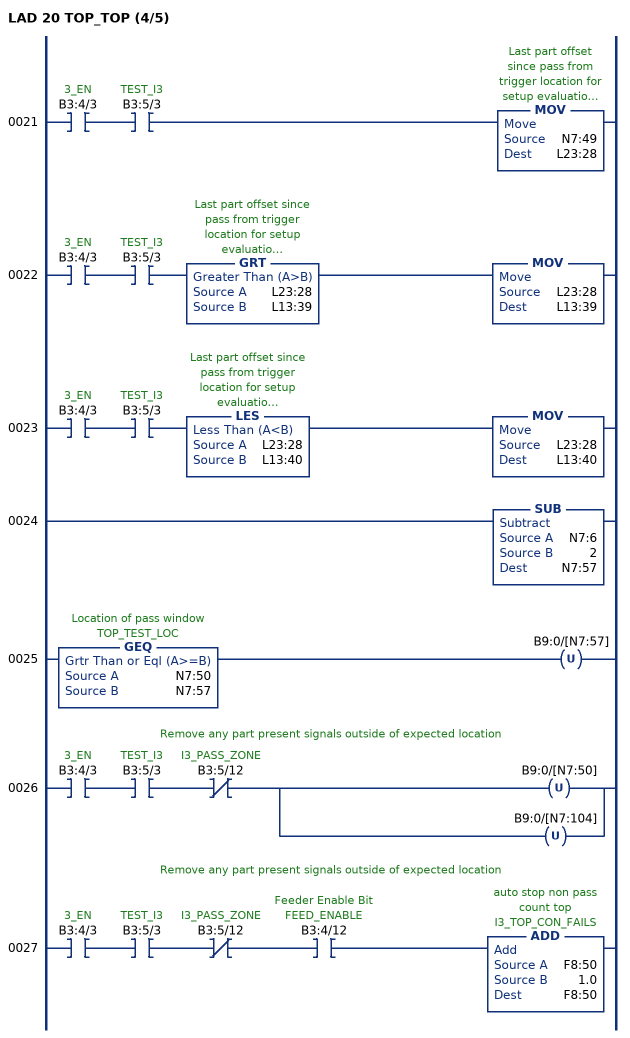
% Rung: 21 %
SOR XIC B3:4/3 XIC B3:5/3 MOV N7:49 L23:28 EOR
%   B3:4/3  3_EN %
%   B3:5/3  TEST_I3 %
%   N7:49  TOP_SINCE_PASS  "distance since top camera pass" %
%   L23:28  LAST_TOP_OFFSET  "Last part offset since pass from trigger location for setup evaluation" %
% Rung: 22 %
SOR XIC B3:4/3 XIC B3:5/3 GRT L23:28 L13:39 MOV L23:28 L13:39 EOR
%   B3:4/3  3_EN %
%   B3:5/3  TEST_I3 %
%   L23:28  LAST_TOP_OFFSET  "Last part offset since pass from trigger location for setup evaluation" %
% Rung: 23 %
SOR XIC B3:4/3 XIC B3:5/3 LES L23:28 L13:40 MOV L23:28 L13:40 EOR
%   B3:4/3  3_EN %
%   B3:5/3  TEST_I3 %
%   L23:28  LAST_TOP_OFFSET  "Last part offset since pass from trigger location for setup evaluation" %
% Rung: 24 %
SOR SUB N7:6 2 N7:57 EOR
%   N7:6  BLOW_LOC_INTEGER  "Blow-off Position" %
% Rung: 25 %
SOR GEQ N7:50 N7:57 OTU B9:0/[N7:57] EOR
%   N7:50  TOP_TEST_LOC  "Location of pass window" %
% Rung: 26 %
% Remove any part present signals outside of expected location %
SOR XIC B3:4/3 XIC B3:5/3 XIO B3:5/12 BST OTU B9:0/[N7:50] NXB OTU B9:0/[N7:104] BND EOR
%   B3:4/3  3_EN %
%   B3:5/3  TEST_I3 %
%   B3:5/12  I3_PASS_ZONE %
%   N7:50  TOP_TEST_LOC  "Location of pass window" %
%   N7:104  2ED_TOP %
% Rung: 27 %
% Remove any part present signals outside of expected location %
SOR XIC B3:4/3 XIC B3:5/3 XIO B3:5/12 XIC B3:4/12 ADD F8:50 1.0 F8:50 EOR
%   B3:4/3  3_EN %
%   B3:5/3  TEST_I3 %
%   B3:5/12  I3_PASS_ZONE %
%   B3:4/12  FEED_ENABLE  "Feeder Enable Bit" %
%   F8:50  I3_TOP_CON_FAILS  "auto stop non pass count top" %

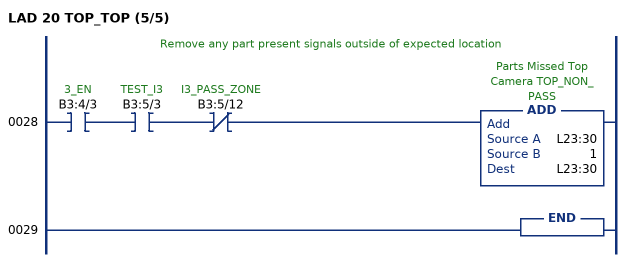
% Rung: 28 %
% Remove any part present signals outside of expected location %
SOR XIC B3:4/3 XIC B3:5/3 XIO B3:5/12 ADD L23:30 1 L23:30 EOR
%   B3:4/3  3_EN %
%   B3:5/3  TEST_I3 %
%   B3:5/12  I3_PASS_ZONE %
%   L23:30  TOP_NON_PASS  "Parts Missed Top Camera" %
% Rung: 29 %
SOR END EOR

LADDER 24 "TOP_BLOW"
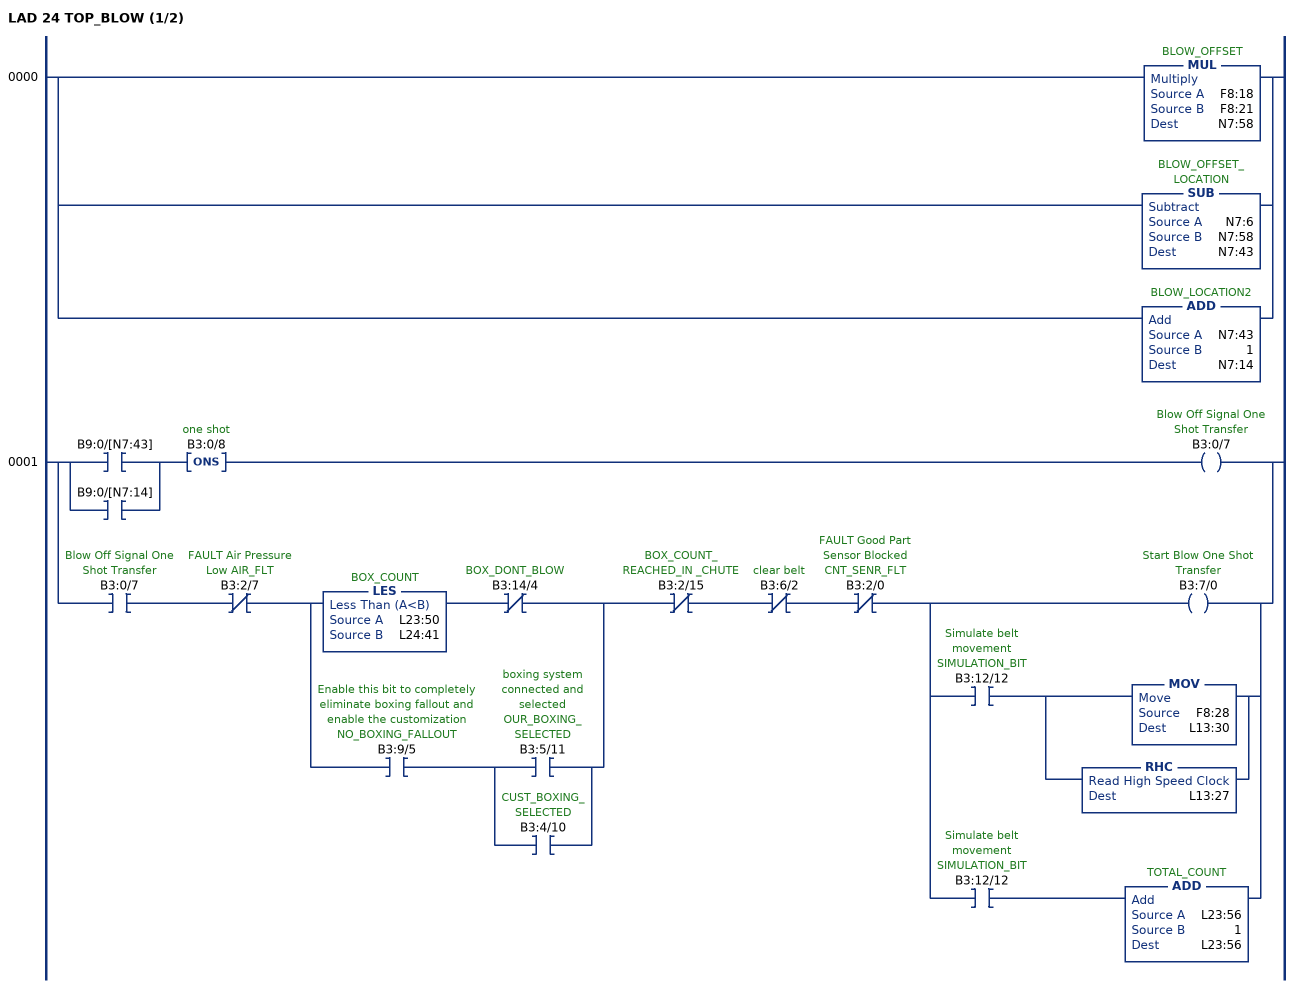
% Rung: 0 %
SOR BST MUL F8:18 F8:21 N7:58 NXB SUB N7:6 N7:58 N7:43 NXB ADD N7:43 1 N7:14 BND EOR
%   F8:18  TOP_SPEED  "top belt speed average in pulses per second 290 Max; Verify" %
%   F8:21  BLOW_COMP_TIME %
%   N7:58  BLOW_OFFSET %
%   N7:6  BLOW_LOC_INTEGER  "Blow-off Position" %
%   N7:43  BLOW_OFFSET_LOCATION %
%   N7:14  BLOW_LOCATION2 %
% Rung: 1 %
SOR BST BST XIC B9:0/[N7:43] NXB XIC B9:0/[N7:14] BND ONS B3:0/8 OTE B3:0/7 NXB XIC B3:0/7 XIO B3:2/7 BST LES L23:50 L24:41 XIO B3:14/4 NXB XIC B3:9/5 BST XIC B3:5/11 NXB XIC B3:4/10 BND BND XIO B3:2/15 XIO B3:6/2 XIO B3:2/0 BST OTE B3:7/0 NXB XIC B3:12/12 BST MOV F8:28 L13:30 NXB RHC L13:27 BND NXB XIC B3:12/12 ADD L23:56 1 L23:56 BND BND EOR
%   N7:43  BLOW_OFFSET_LOCATION %
%   N7:14  BLOW_LOCATION2 %
%   B3:0/8  "one shot" %
%   B3:0/7  "Blow Off Signal One Shot Transfer" %
%   B3:2/7  AIR_FLT  "FAULT Air Pressure Low" %
%   L23:50  BOX_COUNT %
%   L24:41  BOX_COUNT_LIMIT %
%   B3:14/4  BOX_DONT_BLOW %
%   B3:9/5  NO_BOXING_FALLOUT  "Enable this bit to completely eliminate boxing fallout and enable the customization" %
%   B3:5/11  OUR_BOXING_SELECTED  "boxing system connected and selected" %
%   B3:4/10  CUST_BOXING_SELECTED %
%   B3:2/15  "BOX_COUNT_REACHED_IN _CHUTE" %
%   B3:6/2  "clear belt" %
%   B3:2/0  CNT_SENR_FLT  "FAULT Good Part Sensor Blocked" %
%   B3:7/0  "Start Blow One Shot Transfer" %
%   B3:12/12  SIMULATION_BIT  "Simulate belt movement" %
%   F8:28  "momentary rate in ppm" %
%   L23:56  TOTAL_COUNT %

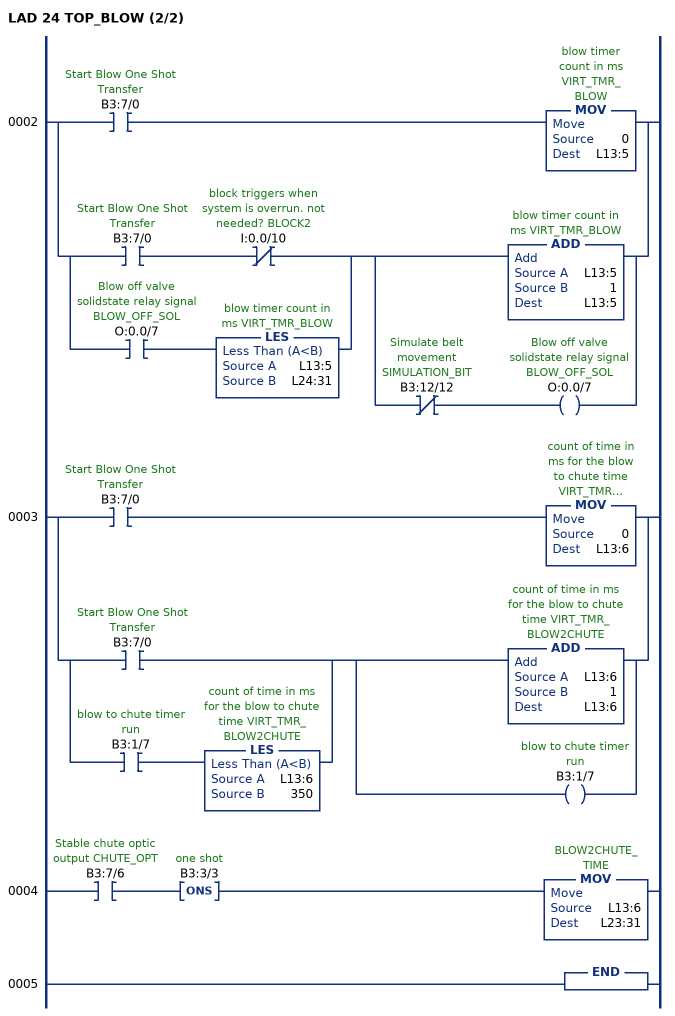
% Rung: 2 %
SOR BST XIC B3:7/0 MOV 0 L13:5 NXB BST XIC B3:7/0 XIO I:0.0/10 NXB XIC O:0.0/7 LES L13:5 L24:31 BND BST ADD L13:5 1 L13:5 NXB XIO B3:12/12 OTE O:0.0/7 BND BND EOR
%   B3:7/0  "Start Blow One Shot Transfer" %
%   L13:5  VIRT_TMR_BLOW  "blow timer count in ms" %
%   I:0.0/10  BLOCK2  "block triggers when system is overrun. not needed?" %
%   O:0.0/7  BLOW_OFF_SOL  "Blow off valve solidstate relay signal" %
%   L24:31  BLOW_TIME %
%   B3:12/12  SIMULATION_BIT  "Simulate belt movement" %
% Rung: 3 %
SOR BST XIC B3:7/0 MOV 0 L13:6 NXB BST XIC B3:7/0 NXB XIC B3:1/7 LES L13:6 350 BND BST ADD L13:6 1 L13:6 NXB OTE B3:1/7 BND BND EOR
%   B3:7/0  "Start Blow One Shot Transfer" %
%   L13:6  VIRT_TMR_BLOW2CHUTE  "count of time in ms for the blow to chute time" %
%   B3:1/7  "blow to chute timer run" %
% Rung: 4 %
SOR XIC B3:7/6 ONS B3:3/3 MOV L13:6 L23:31 EOR
%   B3:7/6  CHUTE_OPT  "Stable chute optic output" %
%   B3:3/3  "one shot" %
%   L13:6  VIRT_TMR_BLOW2CHUTE  "count of time in ms for the blow to chute time" %
%   L23:31  BLOW2CHUTE_TIME %
% Rung: 5 %
SOR END EOR

LADDER 28 "FAULTS"
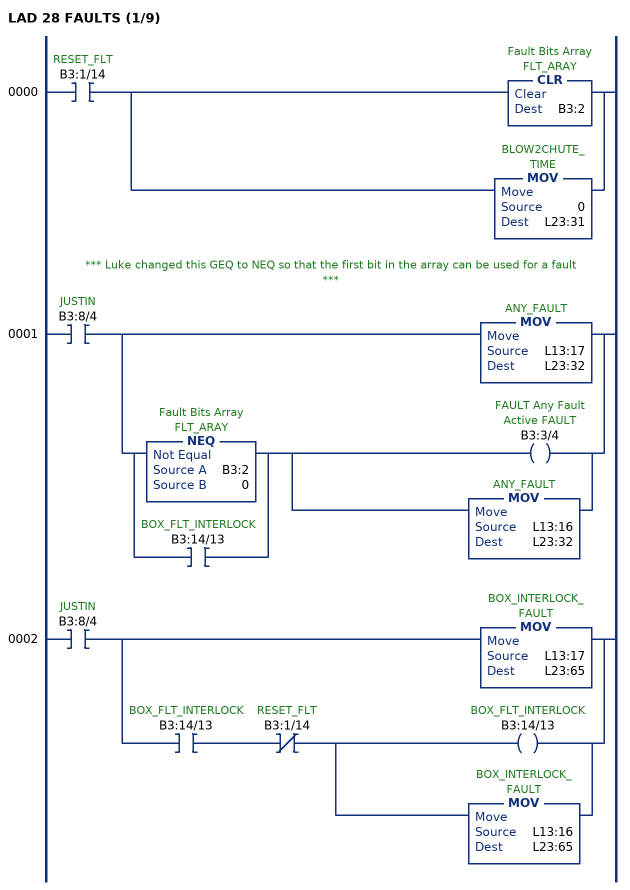
% Rung: 0 %
SOR XIC B3:1/14 BST CLR B3:2 NXB MOV 0 L23:31 BND EOR
%   B3:1/14  RESET_FLT %
%   B3:2  FLT_ARAY  "Fault Bits Array" %
%   L23:31  BLOW2CHUTE_TIME %
% Rung: 1 %
% *** Luke changed this GEQ to NEQ so that the first bit in the array can be used for a fault *** %
SOR XIC B3:8/4 BST MOV L13:17 L23:32 NXB BST NEQ B3:2 0 NXB XIC B3:14/13 BND BST OTE B3:3/4 NXB MOV L13:16 L23:32 BND BND EOR
%   B3:8/4  JUSTIN %
%   L13:17  FALSE %
%   L23:32  ANY_FAULT %
%   B3:2  FLT_ARAY  "Fault Bits Array" %
%   B3:14/13  BOX_FLT_INTERLOCK %
%   B3:3/4  FAULT  "FAULT Any Fault Active" %
%   L13:16  TRUE  "ONE TIME ENABLE FOR THE TIMES WHEN WE FORGET TO RE-ENABLE AFTER SHIPMENT" %
% Rung: 2 %
SOR XIC B3:8/4 BST MOV L13:17 L23:65 NXB XIC B3:14/13 XIO B3:1/14 BST OTE B3:14/13 NXB MOV L13:16 L23:65 BND BND EOR
%   B3:8/4  JUSTIN %
%   L13:17  FALSE %
%   L23:65  BOX_INTERLOCK_FAULT %
%   B3:14/13  BOX_FLT_INTERLOCK %
%   B3:1/14  RESET_FLT %
%   L13:16  TRUE  "ONE TIME ENABLE FOR THE TIMES WHEN WE FORGET TO RE-ENABLE AFTER SHIPMENT" %

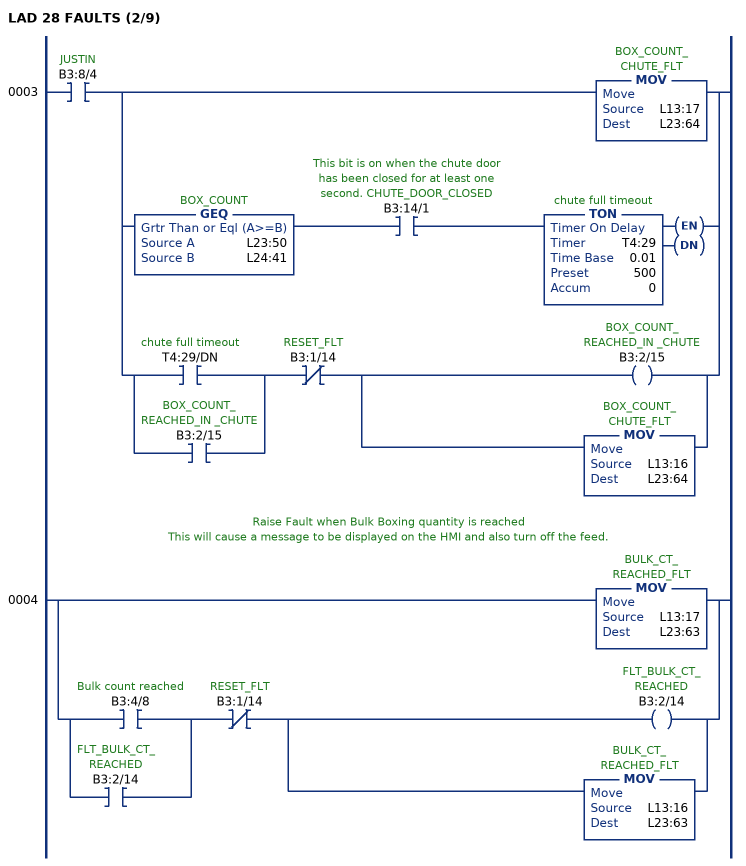
% Rung: 3 %
SOR XIC B3:8/4 BST MOV L13:17 L23:64 NXB GEQ L23:50 L24:41 XIC B3:14/1 TON T4:29 0.01 500 0 NXB BST XIC T4:29/DN NXB XIC B3:2/15 BND XIO B3:1/14 BST OTE B3:2/15 NXB MOV L13:16 L23:64 BND BND EOR
%   B3:8/4  JUSTIN %
%   L13:17  FALSE %
%   L23:64  BOX_COUNT_CHUTE_FLT %
%   L23:50  BOX_COUNT %
%   L24:41  BOX_COUNT_LIMIT %
%   B3:14/1  CHUTE_DOOR_CLOSED  "This bit is on when the chute door has been closed for at least one second." %
%   T4:29  "chute full timeout" %
%   B3:2/15  "BOX_COUNT_REACHED_IN _CHUTE" %
%   B3:1/14  RESET_FLT %
%   L13:16  TRUE  "ONE TIME ENABLE FOR THE TIMES WHEN WE FORGET TO RE-ENABLE AFTER SHIPMENT" %
% Rung: 4 %
% Raise Fault when Bulk Boxing quantity is reached
% 
% This will cause a message to be displayed on the HMI and also turn off the feed. %
SOR BST MOV L13:17 L23:63 NXB BST XIC B3:4/8 NXB XIC B3:2/14 BND XIO B3:1/14 BST OTE B3:2/14 NXB MOV L13:16 L23:63 BND BND EOR
%   L13:17  FALSE %
%   L23:63  BULK_CT_REACHED_FLT %
%   B3:4/8  "Bulk count reached" %
%   B3:2/14  FLT_BULK_CT_REACHED %
%   B3:1/14  RESET_FLT %
%   L13:16  TRUE  "ONE TIME ENABLE FOR THE TIMES WHEN WE FORGET TO RE-ENABLE AFTER SHIPMENT" %

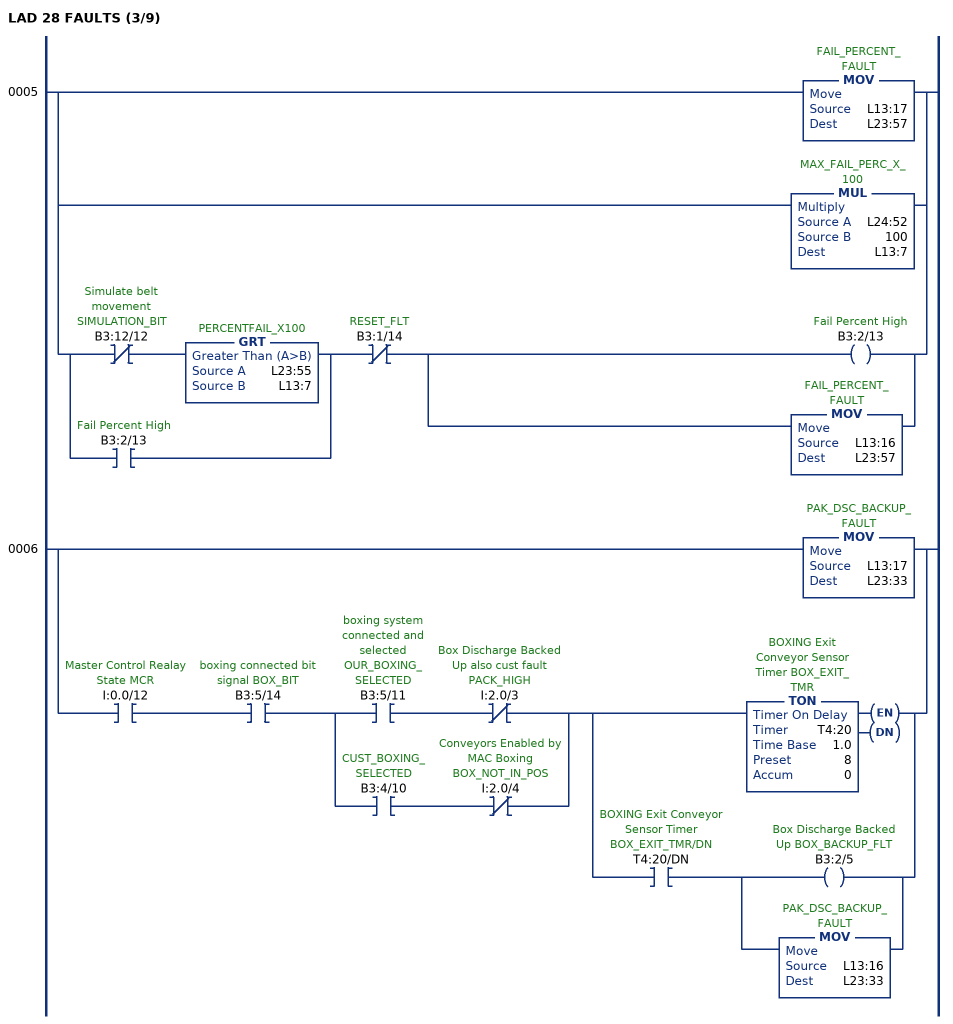
% Rung: 5 %
SOR BST MOV L13:17 L23:57 NXB MUL L24:52 100 L13:7 NXB BST XIO B3:12/12 GRT L23:55 L13:7 NXB XIC B3:2/13 BND XIO B3:1/14 BST OTE B3:2/13 NXB MOV L13:16 L23:57 BND BND EOR
%   L13:17  FALSE %
%   L23:57  FAIL_PERCENT_FAULT %
%   L24:52  MAX_FAIL_PERCENT %
%   L13:7  MAX_FAIL_PERC_X_100 %
%   B3:12/12  SIMULATION_BIT  "Simulate belt movement" %
%   L23:55  PERCENTFAIL_X100 %
%   B3:2/13  "Fail Percent High" %
%   B3:1/14  RESET_FLT %
%   L13:16  TRUE  "ONE TIME ENABLE FOR THE TIMES WHEN WE FORGET TO RE-ENABLE AFTER SHIPMENT" %
% Rung: 6 %
SOR BST MOV L13:17 L23:33 NXB XIC I:0.0/12 XIC B3:5/14 BST XIC B3:5/11 XIO I:2.0/3 NXB XIC B3:4/10 XIO I:2.0/4 BND BST TON T4:20 1.0 8 0 NXB XIC T4:20/DN BST OTE B3:2/5 NXB MOV L13:16 L23:33 BND BND BND EOR
%   L13:17  FALSE %
%   L23:33  PAK_DSC_BACKUP_FAULT %
%   I:0.0/12  MCR  "Master Control Realay State" %
%   B3:5/14  BOX_BIT  "boxing connected bit signal" %
%   B3:5/11  OUR_BOXING_SELECTED  "boxing system connected and selected" %
%   I:2.0/3  PACK_HIGH  "Box Discharge Backed Up also cust fault" %
%   B3:4/10  CUST_BOXING_SELECTED %
%   I:2.0/4  BOX_NOT_IN_POS  "Conveyors Enabled by MAC Boxing" %
%   T4:20  BOX_EXIT_TMR  "BOXING Exit Conveyor Sensor Timer" %
%   B3:2/5  BOX_BACKUP_FLT  "Box Discharge Backed Up" %
%   L13:16  TRUE  "ONE TIME ENABLE FOR THE TIMES WHEN WE FORGET TO RE-ENABLE AFTER SHIPMENT" %

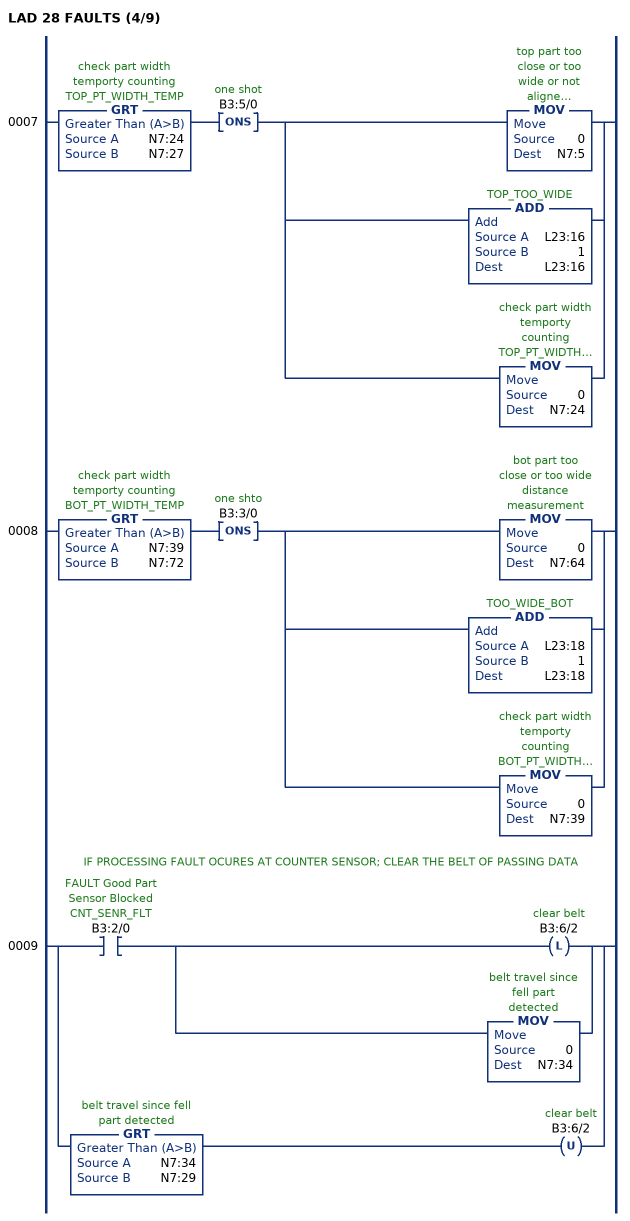
% Rung: 7 %
SOR GRT N7:24 N7:27 ONS B3:5/0 BST MOV 0 N7:5 NXB ADD L23:16 1 L23:16 NXB MOV 0 N7:24 BND EOR
%   N7:24  TOP_PT_WIDTH_TEMP  "check part width temporty counting" %
%   N7:27  "max part width top optic" %
%   B3:5/0  "one shot" %
%   N7:5  "top part too close or too wide or not aligned distance measurement" %
%   L23:16  TOP_TOO_WIDE %
% Rung: 8 %
SOR GRT N7:39 N7:72 ONS B3:3/0 BST MOV 0 N7:64 NXB ADD L23:18 1 L23:18 NXB MOV 0 N7:39 BND EOR
%   N7:39  BOT_PT_WIDTH_TEMP  "check part width temporty counting" %
%   N7:72  "max part width bottom optic" %
%   B3:3/0  "one shto" %
%   N7:64  "bot part too close or too wide distance measurement" %
%   L23:18  TOO_WIDE_BOT %
% Rung: 9 %
% IF PROCESSING FAULT OCURES AT COUNTER SENSOR; CLEAR THE BELT OF PASSING DATA %
SOR BST XIC B3:2/0 BST OTL B3:6/2 NXB MOV 0 N7:34 BND NXB GRT N7:34 N7:29 OTU B3:6/2 BND EOR
%   B3:2/0  CNT_SENR_FLT  "FAULT Good Part Sensor Blocked" %
%   B3:6/2  "clear belt" %
%   N7:34  "belt travel since fell part detected" %
%   N7:29  "belt travel to wipe parts off of belt when fell part detected" %

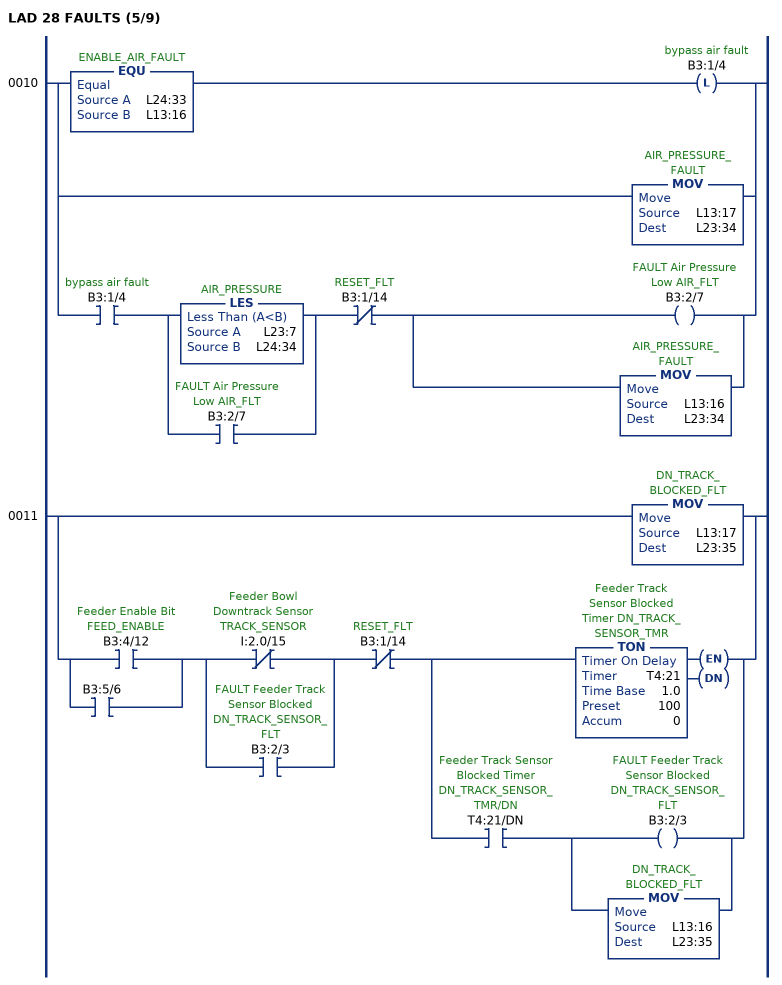
% Rung: 10 %
SOR BST EQU L24:33 L13:16 OTL B3:1/4 NXB MOV L13:17 L23:34 NXB XIC B3:1/4 BST LES L23:7 L24:34 NXB XIC B3:2/7 BND XIO B3:1/14 BST OTE B3:2/7 NXB MOV L13:16 L23:34 BND BND EOR
%   L24:33  ENABLE_AIR_FAULT %
%   L13:16  TRUE  "ONE TIME ENABLE FOR THE TIMES WHEN WE FORGET TO RE-ENABLE AFTER SHIPMENT" %
%   B3:1/4  "bypass air fault" %
%   L13:17  FALSE %
%   L23:34  AIR_PRESSURE_FAULT %
%   L23:7  AIR_PRESSURE %
%   L24:34  MIN_AIR_PRESSURE %
%   B3:2/7  AIR_FLT  "FAULT Air Pressure Low" %
%   B3:1/14  RESET_FLT %
% Rung: 11 %
SOR BST MOV L13:17 L23:35 NXB BST XIC B3:4/12 NXB XIC B3:5/6 BND BST XIO I:2.0/15 NXB XIC B3:2/3 BND XIO B3:1/14 BST TON T4:21 1.0 100 0 NXB XIC T4:21/DN BST OTE B3:2/3 NXB MOV L13:16 L23:35 BND BND BND EOR
%   L13:17  FALSE %
%   L23:35  DN_TRACK_BLOCKED_FLT %
%   B3:4/12  FEED_ENABLE  "Feeder Enable Bit" %
%   I:2.0/15  TRACK_SENSOR  "Feeder Bowl Downtrack Sensor" %
%   B3:2/3  DN_TRACK_SENSOR_FLT  "FAULT Feeder Track Sensor Blocked" %
%   B3:1/14  RESET_FLT %
%   T4:21  DN_TRACK_SENSOR_TMR  "Feeder Track Sensor Blocked Timer" %
%   L13:16  TRUE  "ONE TIME ENABLE FOR THE TIMES WHEN WE FORGET TO RE-ENABLE AFTER SHIPMENT" %

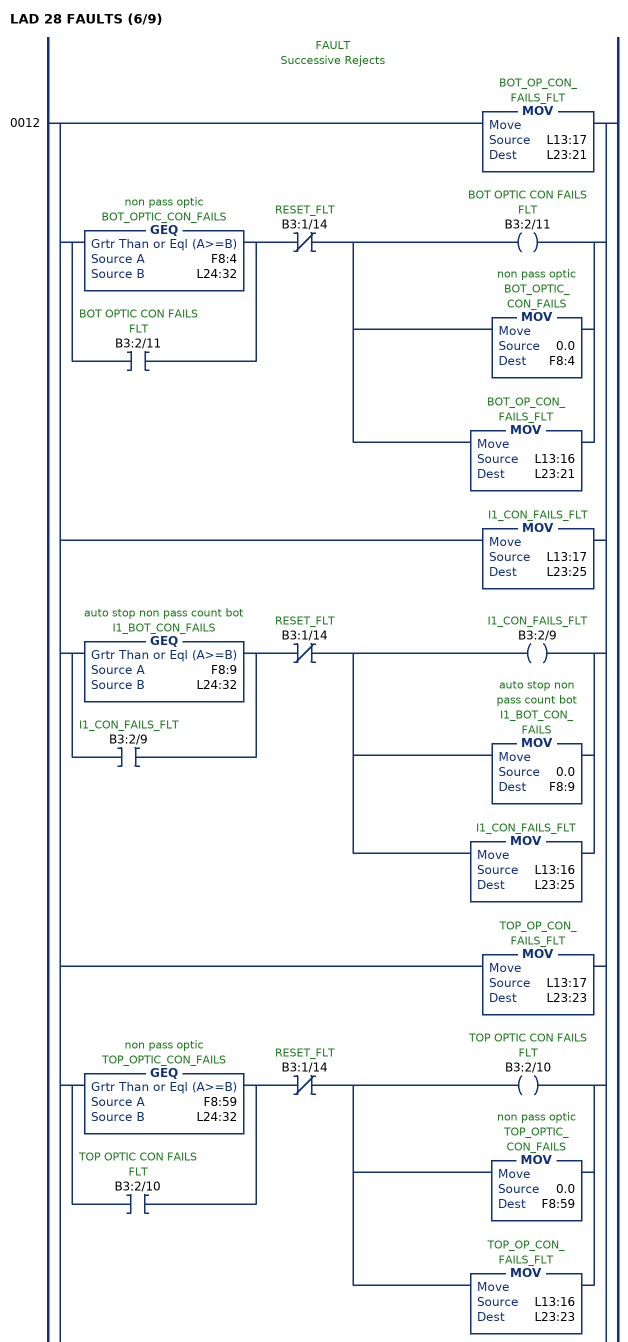

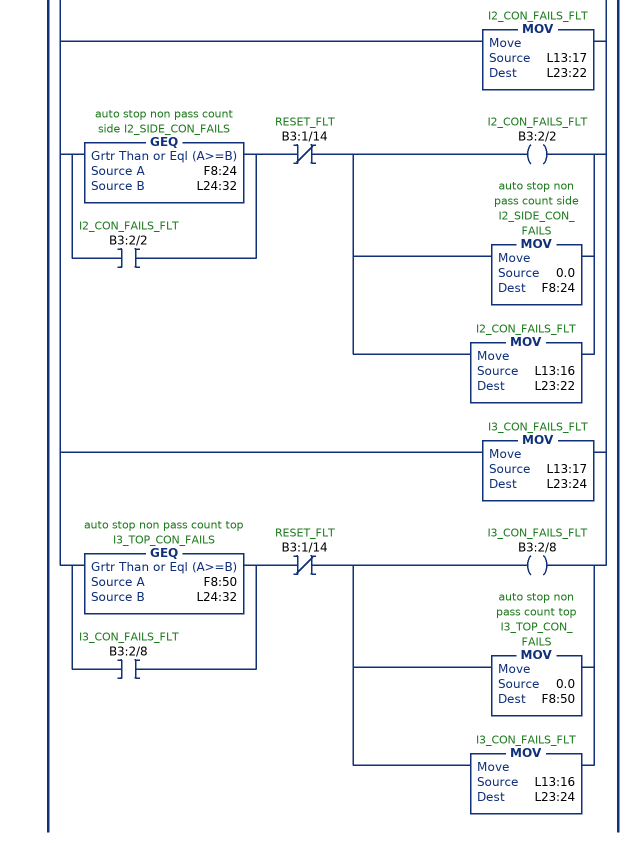
% Rung: 12 %
% FAULT
% Successive Rejects %
SOR BST BST MOV L13:17 L23:21 NXB BST GEQ F8:4 L24:32 NXB XIC B3:2/11 BND XIO B3:1/14 BST OTE B3:2/11 NXB MOV 0.0 F8:4 NXB MOV L13:16 L23:21 BND BND NXB BST MOV L13:17 L23:25 NXB BST GEQ F8:9 L24:32 NXB XIC B3:2/9 BND XIO B3:1/14 BST OTE B3:2/9 NXB MOV 0.0 F8:9 NXB MOV L13:16 L23:25 BND BND NXB BST MOV L13:17 L23:23 NXB BST GEQ F8:59 L24:32 NXB XIC B3:2/10 BND XIO B3:1/14 BST OTE B3:2/10 NXB MOV 0.0 F8:59 NXB MOV L13:16 L23:23 BND BND NXB BST MOV L13:17 L23:22 NXB BST GEQ F8:24 L24:32 NXB XIC B3:2/2 BND XIO B3:1/14 BST OTE B3:2/2 NXB MOV 0.0 F8:24 NXB MOV L13:16 L23:22 BND BND NXB BST MOV L13:17 L23:24 NXB BST GEQ F8:50 L24:32 NXB XIC B3:2/8 BND XIO B3:1/14 BST OTE B3:2/8 NXB MOV 0.0 F8:50 NXB MOV L13:16 L23:24 BND BND BND EOR
%   L13:17  FALSE %
%   L23:21  BOT_OP_CON_FAILS_FLT %
%   F8:4  BOT_OPTIC_CON_FAILS  "non pass optic" %
%   L24:32  MAX_CON_FAILS %
%   B3:2/11  "BOT OPTIC CON FAILS FLT" %
%   B3:1/14  RESET_FLT %
%   L13:16  TRUE  "ONE TIME ENABLE FOR THE TIMES WHEN WE FORGET TO RE-ENABLE AFTER SHIPMENT" %
%   L23:25  I1_CON_FAILS_FLT %
%   F8:9  I1_BOT_CON_FAILS  "auto stop non pass count bot" %
%   B3:2/9  "I1_CON_FAILS_FLT" %
%   L23:23  TOP_OP_CON_FAILS_FLT %
%   F8:59  TOP_OPTIC_CON_FAILS  "non pass optic" %
%   B3:2/10  "TOP OPTIC CON FAILS FLT" %
%   L23:22  I2_CON_FAILS_FLT %
%   F8:24  I2_SIDE_CON_FAILS  "auto stop non pass count side" %
%   B3:2/2  "I2_CON_FAILS_FLT" %
%   L23:24  I3_CON_FAILS_FLT %
%   F8:50  I3_TOP_CON_FAILS  "auto stop non pass count top" %
%   B3:2/8  "I3_CON_FAILS_FLT" %

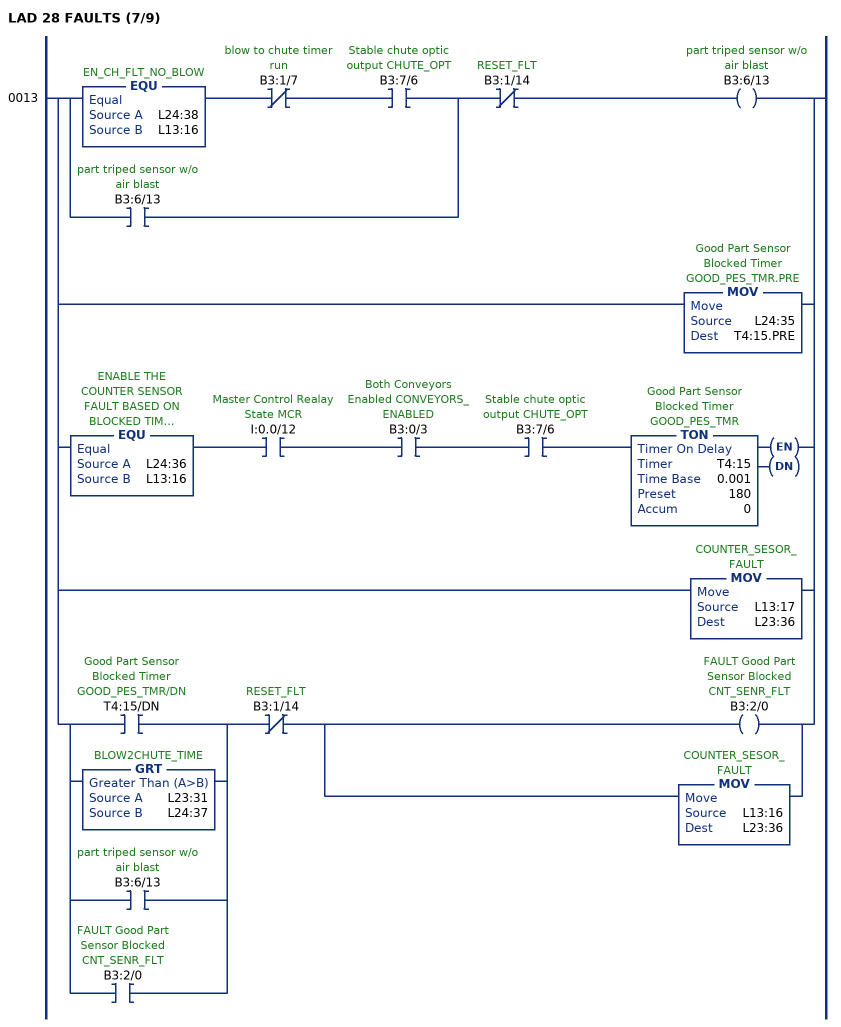
% Rung: 13 %
SOR BST BST EQU L24:38 L13:16 XIO B3:1/7 XIC B3:7/6 NXB XIC B3:6/13 BND XIO B3:1/14 OTE B3:6/13 NXB MOV L24:35 T4:15.PRE NXB EQU L24:36 L13:16 XIC I:0.0/12 XIC B3:0/3 XIC B3:7/6 TON T4:15 0.001 180 0 NXB MOV L13:17 L23:36 NXB BST XIC T4:15/DN NXB GRT L23:31 L24:37 NXB XIC B3:6/13 NXB XIC B3:2/0 BND XIO B3:1/14 BST OTE B3:2/0 NXB MOV L13:16 L23:36 BND BND EOR
%   L24:38  EN_CH_FLT_NO_BLOW %
%   L13:16  TRUE  "ONE TIME ENABLE FOR THE TIMES WHEN WE FORGET TO RE-ENABLE AFTER SHIPMENT" %
%   B3:1/7  "blow to chute timer run" %
%   B3:7/6  CHUTE_OPT  "Stable chute optic output" %
%   B3:6/13  "part triped sensor w/o air blast" %
%   B3:1/14  RESET_FLT %
%   L24:35  GD_PT_SEN_BLKED_TM %
%   T4:15  GOOD_PES_TMR  "Good Part Sensor Blocked Timer" %
%   L24:36  EN_CT_BL_TM_FAULT  "ENABLE THE COUNTER SENSOR FAULT BASED ON BLOCKED TIME" %
%   I:0.0/12  MCR  "Master Control Realay State" %
%   B3:0/3  CONVEYORS_ENABLED  "Both Conveyors Enabled" %
%   L13:17  FALSE %
%   L23:36  COUNTER_SESOR_FAULT %
%   L23:31  BLOW2CHUTE_TIME %
%   L24:37  MAX_BLOW2CHUTE_MS %
%   B3:2/0  CNT_SENR_FLT  "FAULT Good Part Sensor Blocked" %

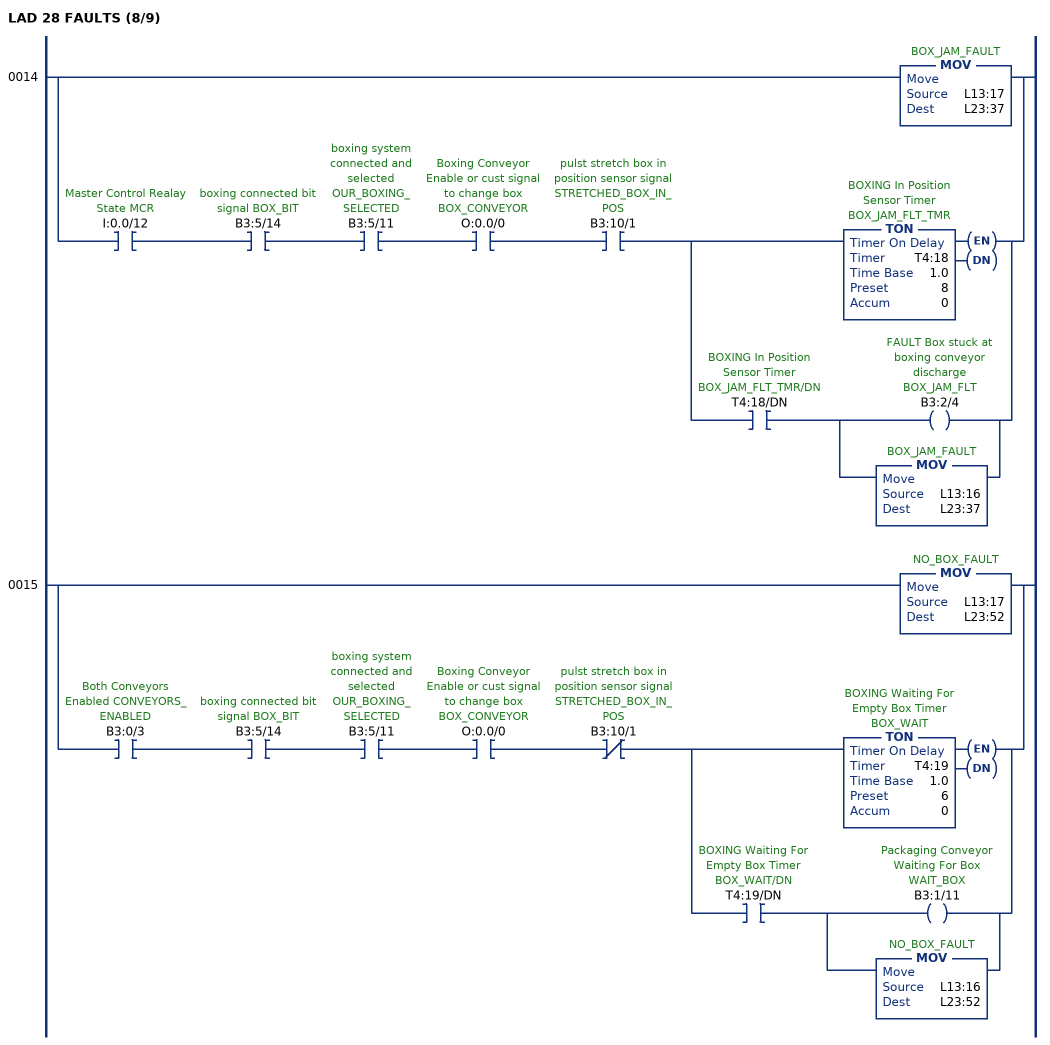
% Rung: 14 %
SOR BST MOV L13:17 L23:37 NXB XIC I:0.0/12 XIC B3:5/14 XIC B3:5/11 XIC O:0.0/0 XIC B3:10/1 BST TON T4:18 1.0 8 0 NXB XIC T4:18/DN BST OTE B3:2/4 NXB MOV L13:16 L23:37 BND BND BND EOR
%   L13:17  FALSE %
%   L23:37  BOX_JAM_FAULT %
%   I:0.0/12  MCR  "Master Control Realay State" %
%   B3:5/14  BOX_BIT  "boxing connected bit signal" %
%   B3:5/11  OUR_BOXING_SELECTED  "boxing system connected and selected" %
%   O:0.0/0  BOX_CONVEYOR  "Boxing Conveyor Enable or cust signal to change box" %
%   B3:10/1  STRETCHED_BOX_IN_POS  "pulst stretch box in position sensor signal" %
%   T4:18  BOX_JAM_FLT_TMR  "BOXING In Position Sensor Timer" %
%   B3:2/4  BOX_JAM_FLT  "FAULT Box stuck at boxing conveyor discharge" %
%   L13:16  TRUE  "ONE TIME ENABLE FOR THE TIMES WHEN WE FORGET TO RE-ENABLE AFTER SHIPMENT" %
% Rung: 15 %
SOR BST MOV L13:17 L23:52 NXB XIC B3:0/3 XIC B3:5/14 XIC B3:5/11 XIC O:0.0/0 XIO B3:10/1 BST TON T4:19 1.0 6 0 NXB XIC T4:19/DN BST OTE B3:1/11 NXB MOV L13:16 L23:52 BND BND BND EOR
%   L13:17  FALSE %
%   L23:52  NO_BOX_FAULT %
%   B3:0/3  CONVEYORS_ENABLED  "Both Conveyors Enabled" %
%   B3:5/14  BOX_BIT  "boxing connected bit signal" %
%   B3:5/11  OUR_BOXING_SELECTED  "boxing system connected and selected" %
%   O:0.0/0  BOX_CONVEYOR  "Boxing Conveyor Enable or cust signal to change box" %
%   B3:10/1  STRETCHED_BOX_IN_POS  "pulst stretch box in position sensor signal" %
%   T4:19  BOX_WAIT  "BOXING Waiting For Empty Box Timer" %
%   B3:1/11  WAIT_BOX  "Packaging Conveyor Waiting For Box" %
%   L13:16  TRUE  "ONE TIME ENABLE FOR THE TIMES WHEN WE FORGET TO RE-ENABLE AFTER SHIPMENT" %

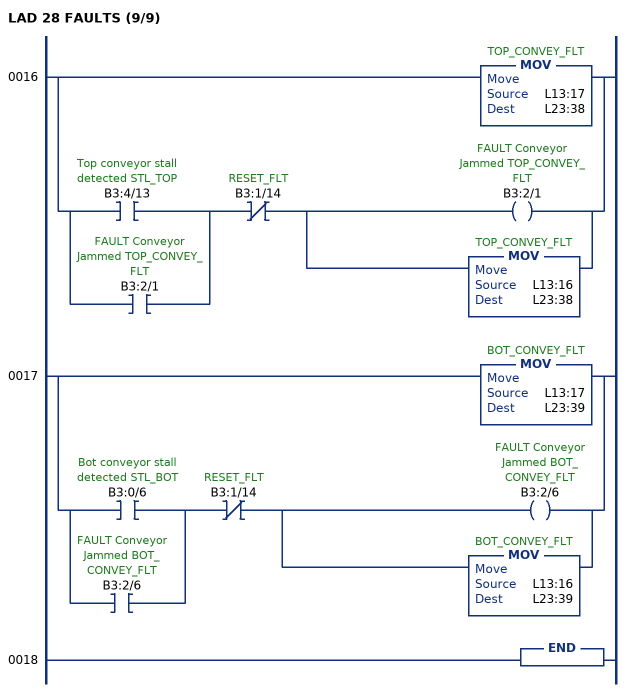
% Rung: 16 %
SOR BST MOV L13:17 L23:38 NXB BST XIC B3:4/13 NXB XIC B3:2/1 BND XIO B3:1/14 BST OTE B3:2/1 NXB MOV L13:16 L23:38 BND BND EOR
%   L13:17  FALSE %
%   L23:38  TOP_CONVEY_FLT %
%   B3:4/13  STL_TOP  "Top conveyor stall detected" %
%   B3:2/1  "FAULT Conveyor Jammed TOP_CONVEY_FLT" %
%   B3:1/14  RESET_FLT %
%   L13:16  TRUE  "ONE TIME ENABLE FOR THE TIMES WHEN WE FORGET TO RE-ENABLE AFTER SHIPMENT" %
% Rung: 17 %
SOR BST MOV L13:17 L23:39 NXB BST XIC B3:0/6 NXB XIC B3:2/6 BND XIO B3:1/14 BST OTE B3:2/6 NXB MOV L13:16 L23:39 BND BND EOR
%   L13:17  FALSE %
%   L23:39  BOT_CONVEY_FLT %
%   B3:0/6  STL_BOT  "Bot conveyor stall detected" %
%   B3:2/6  "FAULT Conveyor Jammed BOT_CONVEY_FLT" %
%   B3:1/14  RESET_FLT %
%   L13:16  TRUE  "ONE TIME ENABLE FOR THE TIMES WHEN WE FORGET TO RE-ENABLE AFTER SHIPMENT" %
% Rung: 18 %
SOR END EOR

LADDER 29 "SPEED"
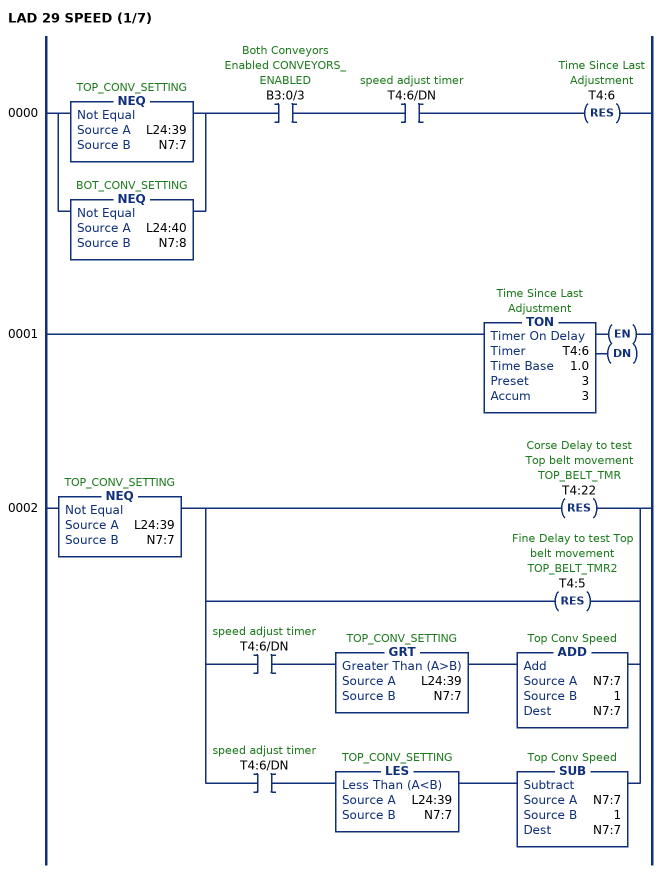
% Rung: 0 %
SOR BST NEQ L24:39 N7:7 NXB NEQ L24:40 N7:8 BND XIC B3:0/3 XIC T4:6/DN RES T4:6 EOR
%   L24:39  TOP_CONV_SETTING %
%   N7:7  "Top Conv Speed" %
%   L24:40  BOT_CONV_SETTING %
%   N7:8  "Bottom Conveyor Speed" %
%   B3:0/3  CONVEYORS_ENABLED  "Both Conveyors Enabled" %
%   T4:6/DN  "speed adjust timer" %
%   T4:6  "Time Since Last Adjustment" %
% Rung: 1 %
SOR TON T4:6 1.0 3 3 EOR
%   T4:6  "Time Since Last Adjustment" %
% Rung: 2 %
SOR NEQ L24:39 N7:7 BST RES T4:22 NXB RES T4:5 NXB XIC T4:6/DN GRT L24:39 N7:7 ADD N7:7 1 N7:7 NXB XIC T4:6/DN LES L24:39 N7:7 SUB N7:7 1 N7:7 BND EOR
%   L24:39  TOP_CONV_SETTING %
%   N7:7  "Top Conv Speed" %
%   T4:22  TOP_BELT_TMR  "Corse Delay to test Top belt movement" %
%   T4:5  TOP_BELT_TMR2  "Fine Delay to test Top belt movement" %
%   T4:6/DN  "speed adjust timer" %

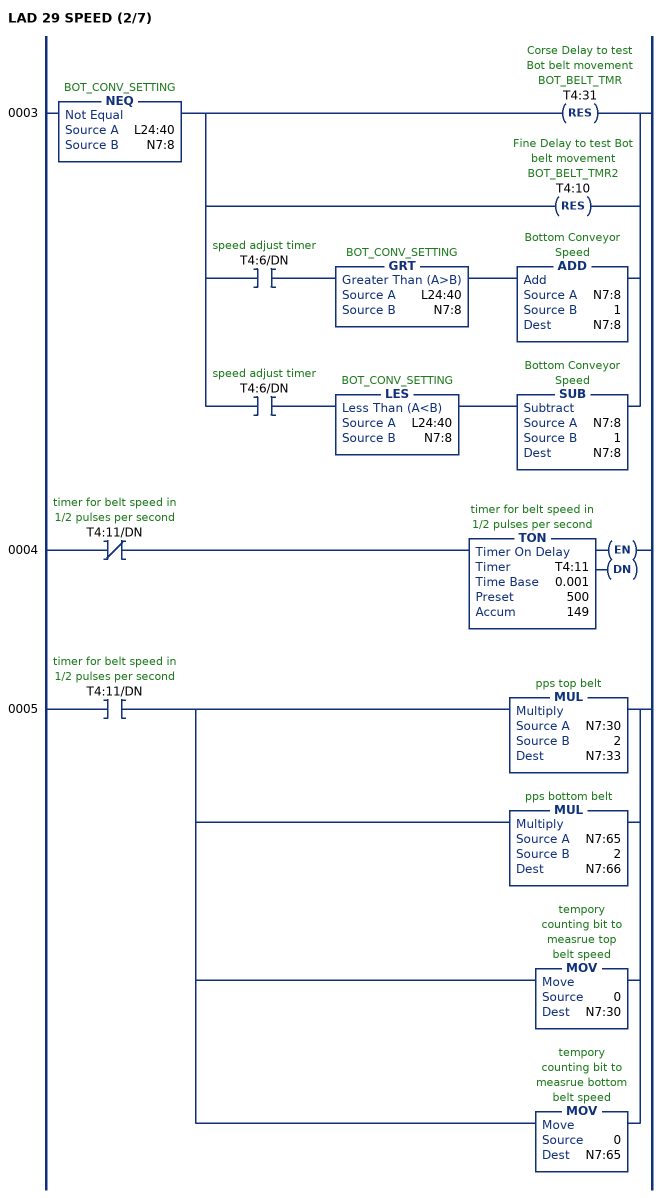
% Rung: 3 %
SOR NEQ L24:40 N7:8 BST RES T4:31 NXB RES T4:10 NXB XIC T4:6/DN GRT L24:40 N7:8 ADD N7:8 1 N7:8 NXB XIC T4:6/DN LES L24:40 N7:8 SUB N7:8 1 N7:8 BND EOR
%   L24:40  BOT_CONV_SETTING %
%   N7:8  "Bottom Conveyor Speed" %
%   T4:31  BOT_BELT_TMR  "Corse Delay to test Bot belt movement" %
%   T4:10  BOT_BELT_TMR2  "Fine Delay to test Bot belt movement" %
%   T4:6/DN  "speed adjust timer" %
% Rung: 4 %
SOR XIO T4:11/DN TON T4:11 0.001 500 149 EOR
%   T4:11  "timer for belt speed in 1/2 pulses per second" %
% Rung: 5 %
SOR XIC T4:11/DN BST MUL N7:30 2 N7:33 NXB MUL N7:65 2 N7:66 NXB MOV 0 N7:30 NXB MOV 0 N7:65 BND EOR
%   T4:11  "timer for belt speed in 1/2 pulses per second" %
%   N7:30  "tempory counting bit to measrue top belt speed" %
%   N7:33  "pps top belt" %
%   N7:65  "tempory counting bit to measrue bottom belt speed" %
%   N7:66  "pps bottom belt" %

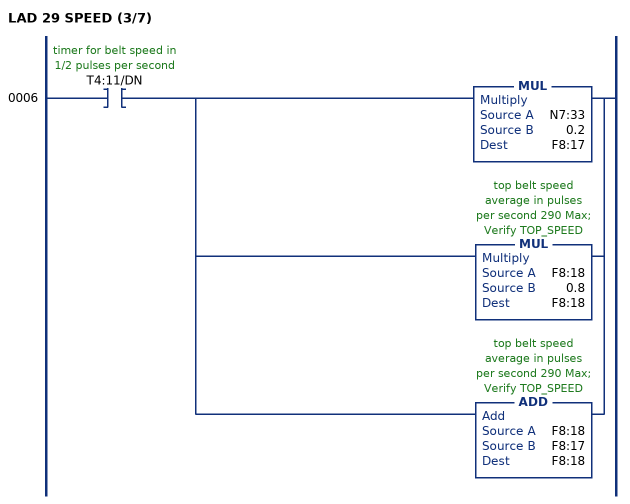
% Rung: 6 %
SOR XIC T4:11/DN BST MUL N7:33 0.2 F8:17 NXB MUL F8:18 0.8 F8:18 NXB ADD F8:18 F8:17 F8:18 BND EOR
%   T4:11  "timer for belt speed in 1/2 pulses per second" %
%   N7:33  "pps top belt" %
%   F8:18  TOP_SPEED  "top belt speed average in pulses per second 290 Max; Verify" %

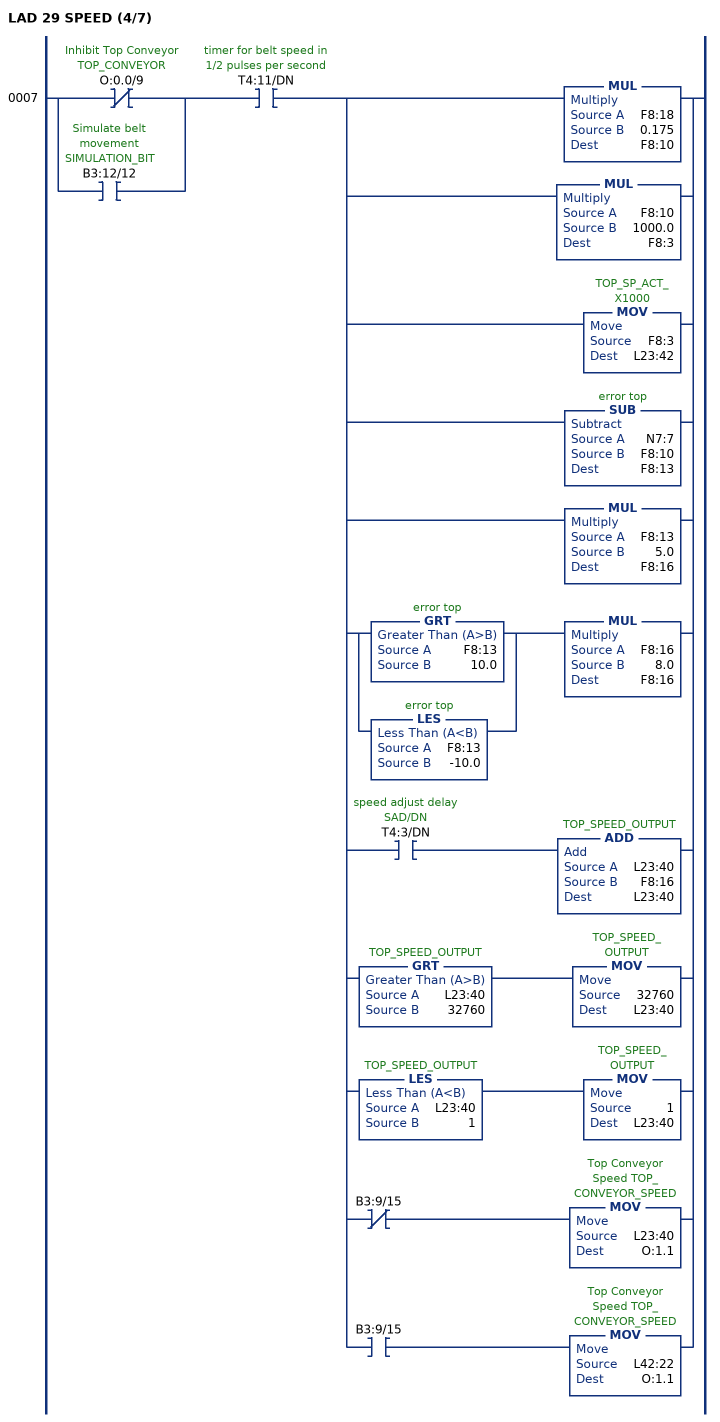
% Rung: 7 %
SOR BST XIO O:0.0/9 NXB XIC B3:12/12 BND XIC T4:11/DN BST MUL F8:18 0.175 F8:10 NXB MUL F8:10 1000.0 F8:3 NXB MOV F8:3 L23:42 NXB SUB N7:7 F8:10 F8:13 NXB MUL F8:13 5.0 F8:16 NXB BST GRT F8:13 10.0 NXB LES F8:13 -10.0 BND MUL F8:16 8.0 F8:16 NXB XIC T4:3/DN ADD L23:40 F8:16 L23:40 NXB GRT L23:40 32760 MOV 32760 L23:40 NXB LES L23:40 1 MOV 1 L23:40 NXB XIO B3:9/15 MOV L23:40 O:1.1 NXB XIC B3:9/15 MOV L42:22 O:1.1 BND EOR
%   O:0.0/9  TOP_CONVEYOR  "Inhibit Top Conveyor" %
%   B3:12/12  SIMULATION_BIT  "Simulate belt movement" %
%   T4:11  "timer for belt speed in 1/2 pulses per second" %
%   F8:18  TOP_SPEED  "top belt speed average in pulses per second 290 Max; Verify" %
%   L23:42  TOP_SP_ACT_X1000 %
%   N7:7  "Top Conv Speed" %
%   F8:13  "error top" %
%   T4:3  SAD  "speed adjust delay" %
%   L23:40  TOP_SPEED_OUTPUT %
%   O:1.1  TOP_CONVEYOR_SPEED  "Top Conveyor Speed" %

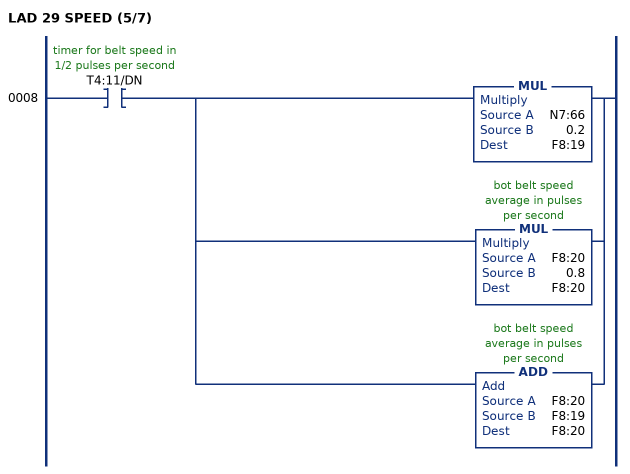
% Rung: 8 %
SOR XIC T4:11/DN BST MUL N7:66 0.2 F8:19 NXB MUL F8:20 0.8 F8:20 NXB ADD F8:20 F8:19 F8:20 BND EOR
%   T4:11  "timer for belt speed in 1/2 pulses per second" %
%   N7:66  "pps bottom belt" %
%   F8:20  "bot belt speed average in pulses per second" %

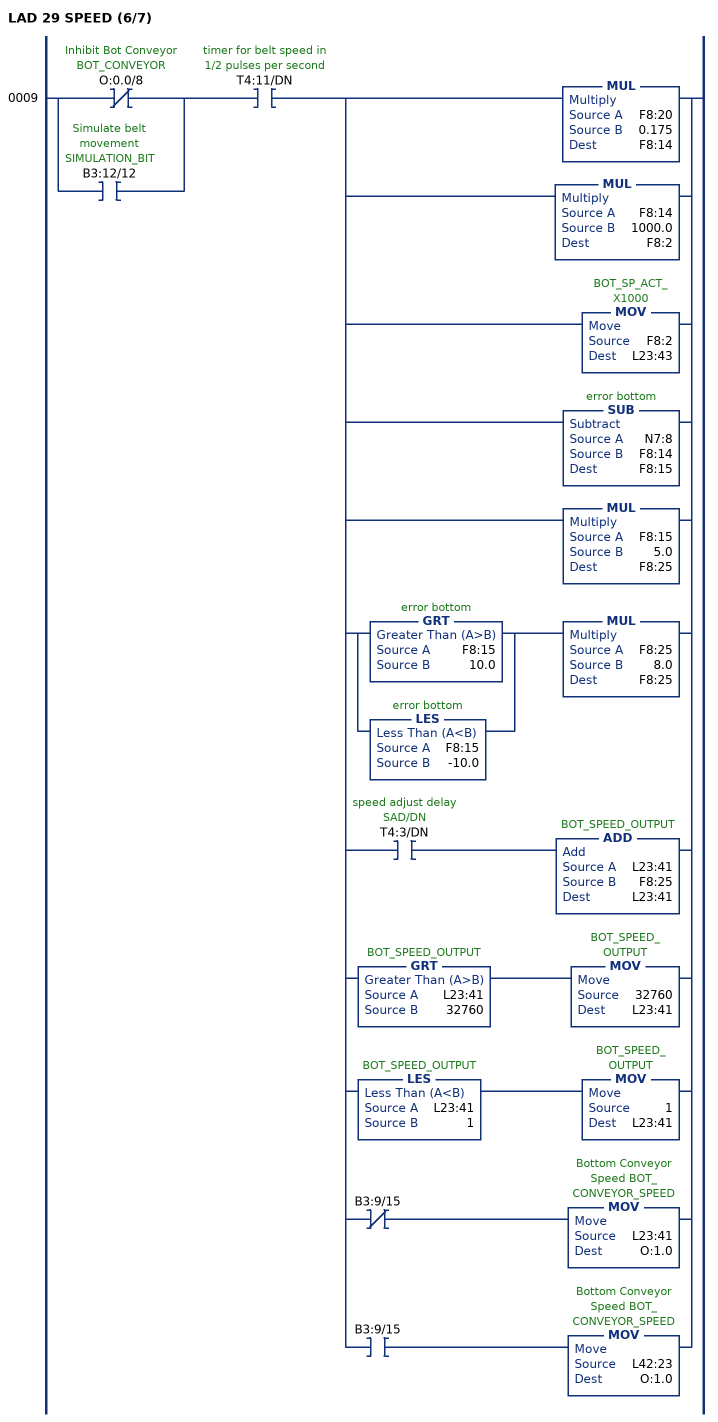
% Rung: 9 %
SOR BST XIO O:0.0/8 NXB XIC B3:12/12 BND XIC T4:11/DN BST MUL F8:20 0.175 F8:14 NXB MUL F8:14 1000.0 F8:2 NXB MOV F8:2 L23:43 NXB SUB N7:8 F8:14 F8:15 NXB MUL F8:15 5.0 F8:25 NXB BST GRT F8:15 10.0 NXB LES F8:15 -10.0 BND MUL F8:25 8.0 F8:25 NXB XIC T4:3/DN ADD L23:41 F8:25 L23:41 NXB GRT L23:41 32760 MOV 32760 L23:41 NXB LES L23:41 1 MOV 1 L23:41 NXB XIO B3:9/15 MOV L23:41 O:1.0 NXB XIC B3:9/15 MOV L42:23 O:1.0 BND EOR
%   O:0.0/8  BOT_CONVEYOR  "Inhibit Bot Conveyor" %
%   B3:12/12  SIMULATION_BIT  "Simulate belt movement" %
%   T4:11  "timer for belt speed in 1/2 pulses per second" %
%   F8:20  "bot belt speed average in pulses per second" %
%   L23:43  BOT_SP_ACT_X1000 %
%   N7:8  "Bottom Conveyor Speed" %
%   F8:15  "error bottom" %
%   T4:3  SAD  "speed adjust delay" %
%   L23:41  BOT_SPEED_OUTPUT %
%   O:1.0  BOT_CONVEYOR_SPEED  "Bottom Conveyor Speed" %

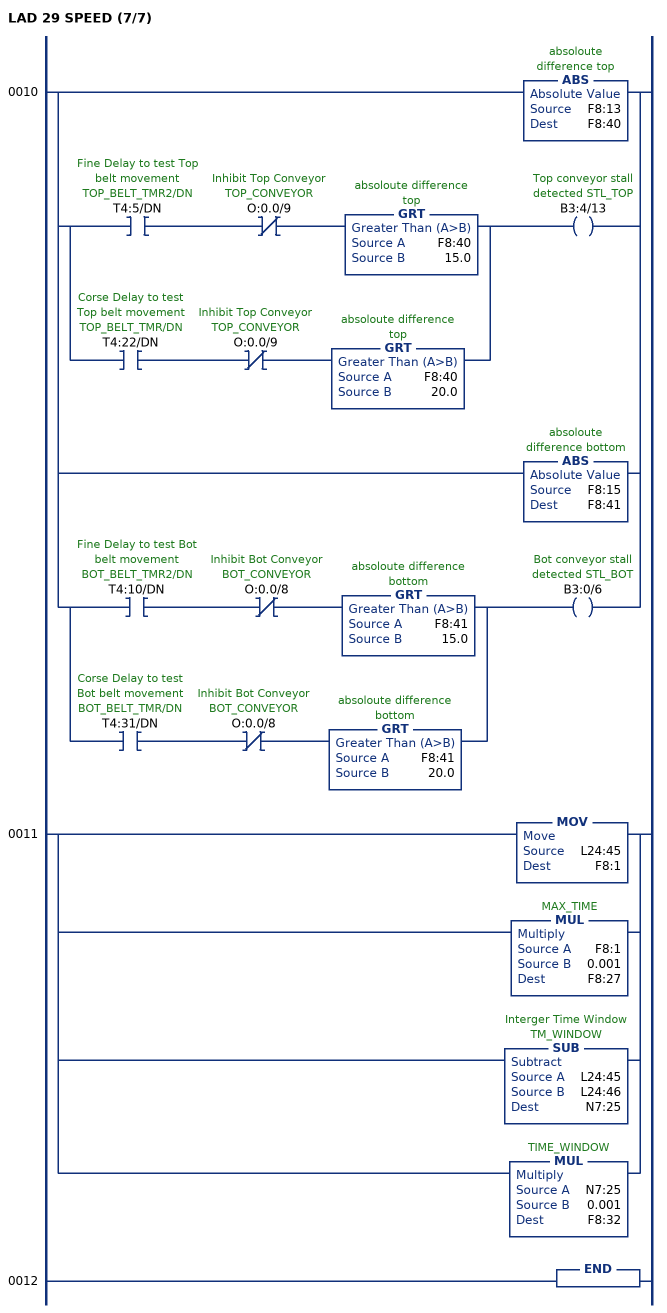
% Rung: 10 %
SOR BST ABS F8:13 F8:40 NXB BST XIC T4:5/DN XIO O:0.0/9 GRT F8:40 15.0 NXB XIC T4:22/DN XIO O:0.0/9 GRT F8:40 20.0 BND OTE B3:4/13 NXB ABS F8:15 F8:41 NXB BST XIC T4:10/DN XIO O:0.0/8 GRT F8:41 15.0 NXB XIC T4:31/DN XIO O:0.0/8 GRT F8:41 20.0 BND OTE B3:0/6 BND EOR
%   F8:13  "error top" %
%   F8:40  "absoloute difference top" %
%   T4:5  TOP_BELT_TMR2  "Fine Delay to test Top belt movement" %
%   O:0.0/9  TOP_CONVEYOR  "Inhibit Top Conveyor" %
%   T4:22  TOP_BELT_TMR  "Corse Delay to test Top belt movement" %
%   B3:4/13  STL_TOP  "Top conveyor stall detected" %
%   F8:15  "error bottom" %
%   F8:41  "absoloute difference bottom" %
%   T4:10  BOT_BELT_TMR2  "Fine Delay to test Bot belt movement" %
%   O:0.0/8  BOT_CONVEYOR  "Inhibit Bot Conveyor" %
%   T4:31  BOT_BELT_TMR  "Corse Delay to test Bot belt movement" %
%   B3:0/6  STL_BOT  "Bot conveyor stall detected" %
% Rung: 11 %
SOR BST MOV L24:45 F8:1 NXB MUL F8:1 0.001 F8:27 NXB SUB L24:45 L24:46 N7:25 NXB MUL N7:25 0.001 F8:32 BND EOR
%   L24:45  VISION_MAX_RES_TIME %
%   F8:27  MAX_TIME %
%   L24:46  VISION_MIN_RES_TIME %
%   N7:25  TM_WINDOW  "Interger Time Window" %
%   F8:32  TIME_WINDOW %
% Rung: 12 %
SOR END EOR

LADDER 30 "COUNT"
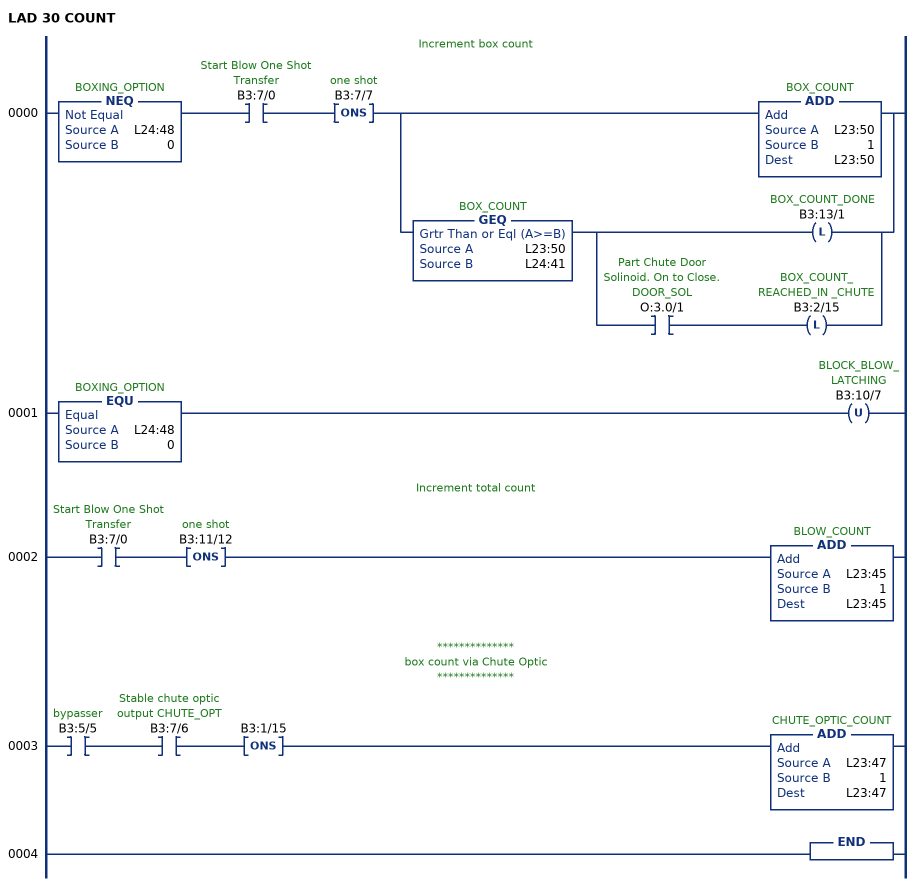
% Rung: 0 %
% Increment box count %
SOR NEQ L24:48 0 XIC B3:7/0 ONS B3:7/7 BST ADD L23:50 1 L23:50 NXB GEQ L23:50 L24:41 BST OTL B3:13/1 NXB XIC O:3.0/1 OTL B3:2/15 BND BND EOR
%   L24:48  BOXING_OPTION %
%   B3:7/0  "Start Blow One Shot Transfer" %
%   B3:7/7  "one shot" %
%   L23:50  BOX_COUNT %
%   L24:41  BOX_COUNT_LIMIT %
%   B3:13/1  BOX_COUNT_DONE %
%   O:3.0/1  DOOR_SOL  "Part Chute Door Solinoid. On to Close." %
%   B3:2/15  "BOX_COUNT_REACHED_IN _CHUTE" %
% Rung: 1 %
SOR EQU L24:48 0 OTU B3:10/7 EOR
%   L24:48  BOXING_OPTION %
%   B3:10/7  BLOCK_BLOW_LATCHING %
% Rung: 2 %
% Increment total count %
SOR XIC B3:7/0 ONS B3:11/12 ADD L23:45 1 L23:45 EOR
%   B3:7/0  "Start Blow One Shot Transfer" %
%   B3:11/12  "one shot" %
%   L23:45  BLOW_COUNT %
% Rung: 3 %
% **************
% box count via Chute Optic
% ************** %
SOR XIC B3:5/5 XIC B3:7/6 ONS B3:1/15 ADD L23:47 1 L23:47 EOR
%   B3:5/5  "bypasser" %
%   B3:7/6  CHUTE_OPT  "Stable chute optic output" %
%   L23:47  CHUTE_OPTIC_COUNT %
% Rung: 4 %
SOR END EOR

LADDER 32 "LINEABOXER"
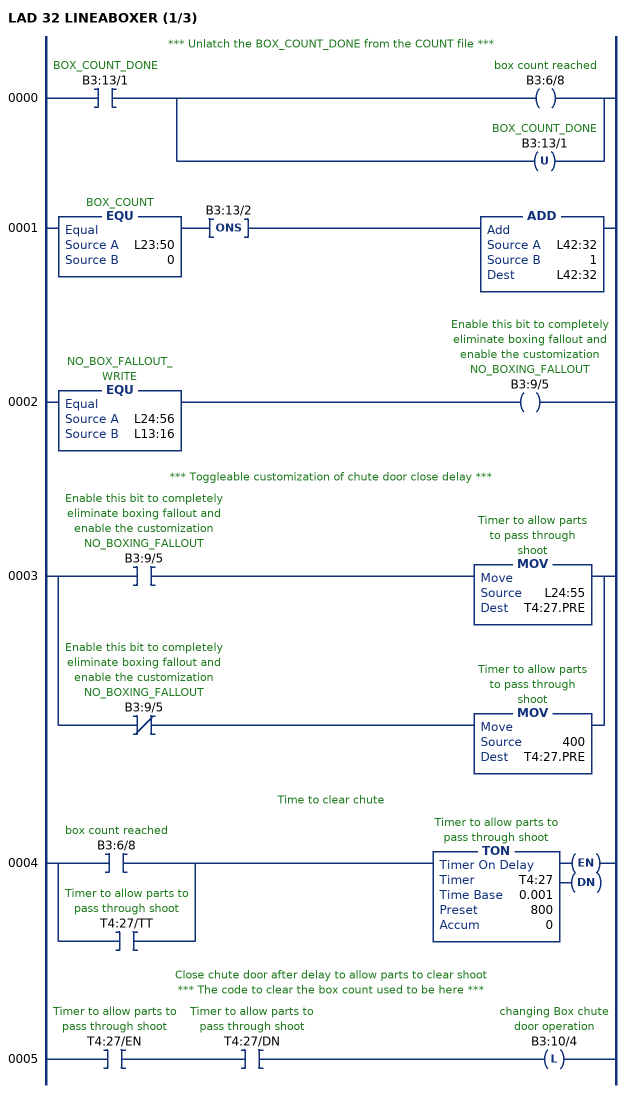
% Rung: 0 %
% *** Unlatch the BOX_COUNT_DONE from the COUNT file *** %
SOR XIC B3:13/1 BST OTE B3:6/8 NXB OTU B3:13/1 BND EOR
%   B3:13/1  BOX_COUNT_DONE %
%   B3:6/8  "box count reached" %
% Rung: 1 %
SOR EQU L23:50 0 ONS B3:13/2 ADD L42:32 1 L42:32 EOR
%   L23:50  BOX_COUNT %
% Rung: 2 %
SOR EQU L24:56 L13:16 OTE B3:9/5 EOR
%   L24:56  NO_BOX_FALLOUT_WRITE %
%   L13:16  TRUE  "ONE TIME ENABLE FOR THE TIMES WHEN WE FORGET TO RE-ENABLE AFTER SHIPMENT" %
%   B3:9/5  NO_BOXING_FALLOUT  "Enable this bit to completely eliminate boxing fallout and enable the customization" %
% Rung: 3 %
% *** Toggleable customization of chute door close delay *** %
SOR BST XIC B3:9/5 MOV L24:55 T4:27.PRE NXB XIO B3:9/5 MOV 400 T4:27.PRE BND EOR
%   B3:9/5  NO_BOXING_FALLOUT  "Enable this bit to completely eliminate boxing fallout and enable the customization" %
%   L24:55  CHUTE_CLOSE_DELAY  "Timer to allow parts to pass through the chute" %
%   T4:27  "Timer to allow parts to pass through shoot" %
% Rung: 4 %
% Time to clear chute %
SOR BST XIC B3:6/8 NXB XIC T4:27/TT BND TON T4:27 0.001 800 0 EOR
%   B3:6/8  "box count reached" %
%   T4:27  "Timer to allow parts to pass through shoot" %
% Rung: 5 %
% Close chute door after delay to allow parts to clear shoot
% *** The code to clear the box count used to be here *** %
SOR XIC T4:27/EN XIC T4:27/DN OTL B3:10/4 EOR
%   T4:27  "Timer to allow parts to pass through shoot" %
%   B3:10/4  "changing Box chute door operation" %

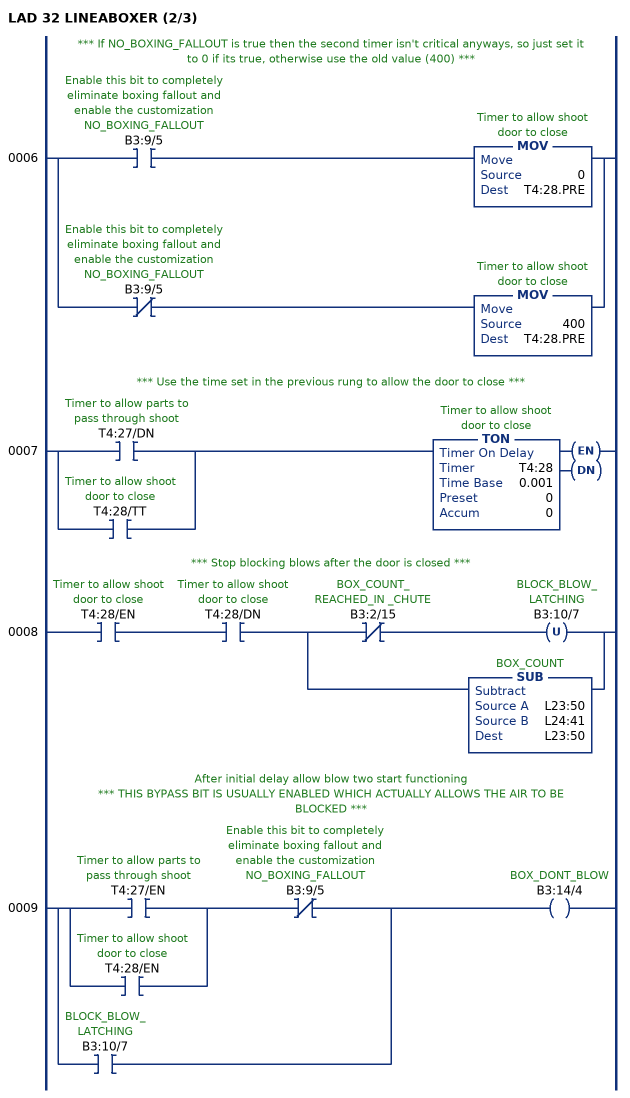
% Rung: 6 %
% *** If NO_BOXING_FALLOUT is true then the second timer isn't critical anyways, so just set it to 0 if its true, otherwise use the old value (400) *** %
SOR BST XIC B3:9/5 MOV 0 T4:28.PRE NXB XIO B3:9/5 MOV 400 T4:28.PRE BND EOR
%   B3:9/5  NO_BOXING_FALLOUT  "Enable this bit to completely eliminate boxing fallout and enable the customization" %
%   T4:28  "Timer to allow shoot door to close" %
% Rung: 7 %
% *** Use the time set in the previous rung to allow the door to close *** %
SOR BST XIC T4:27/DN NXB XIC T4:28/TT BND TON T4:28 0.001 0 0 EOR
%   T4:27  "Timer to allow parts to pass through shoot" %
%   T4:28  "Timer to allow shoot door to close" %
% Rung: 8 %
% *** Stop blocking blows after the door is closed *** %
SOR XIC T4:28/EN XIC T4:28/DN BST XIO B3:2/15 OTU B3:10/7 NXB SUB L23:50 L24:41 L23:50 BND EOR
%   T4:28  "Timer to allow shoot door to close" %
%   B3:2/15  "BOX_COUNT_REACHED_IN _CHUTE" %
%   B3:10/7  BLOCK_BLOW_LATCHING %
%   L23:50  BOX_COUNT %
%   L24:41  BOX_COUNT_LIMIT %
% Rung: 9 %
% After initial delay allow blow two start functioning
% *** THIS BYPASS BIT IS USUALLY ENABLED WHICH ACTUALLY ALLOWS THE AIR TO BE BLOCKED *** %
SOR BST BST XIC T4:27/EN NXB XIC T4:28/EN BND XIO B3:9/5 NXB XIC B3:10/7 BND OTE B3:14/4 EOR
%   T4:27  "Timer to allow parts to pass through shoot" %
%   T4:28  "Timer to allow shoot door to close" %
%   B3:9/5  NO_BOXING_FALLOUT  "Enable this bit to completely eliminate boxing fallout and enable the customization" %
%   B3:10/7  BLOCK_BLOW_LATCHING %
%   B3:14/4  BOX_DONT_BLOW %

